PROGRAM MAIN
VAR
END_VAR

(* 
	GOF 		Provide an interface for creating families of related or dependent objects without
				specifying their concrete classes.
*)
P_AbstractFactory();

END_PROGRAM

(* stored: Version 1.1.0.1, ProductVersion 3.1.4024.12
   POU MAIN: Id {a3eafa91-ed4b-4c56-85b3-699034de4110}, SpecialFunc None *)
